{attribute 'qualified_only'}
VAR_GLOBAL
END_VAR

(* stored: Version 1.1.0.1, ProductVersion 3.1.4022.7
   GVL GVL_06_Output_Other: Id {f85a2549-003a-4bd6-b846-a049b0b1aaa3} *)
